FUNCTION SAFE_MEMCPY : BOOL

VAR_INPUT
	pDst : POINTER TO BYTE;
	nDstLen : UDINT;
	pSrc : POINTER TO BYTE;
	nSrcLen : UDINT;
END_VAR

VAR
	nMcErr : UDINT;
END_VAR

IF nDstLen < nSrcLen THEN
	SAFE_MEMCPY := FALSE;
END_IF

nMcErr := MEMCPY(pDst, pSrc, nSrcLen);
IF nMcErr = 0 THEN
	SAFE_MEMCPY := FALSE;
END_IF

SAFE_MEMCPY := TRUE;

END_FUNCTION

(* stored: Version 1.1.0.1
   POU SAFE_MEMCPY: Id {7c59690b-5c27-4eac-81b1-0f5b54aa1407}, SpecialFunc None *)
